INTERFACE I_Cyl_Diag

METHOD M_Diag : E_Diag
VAR_INPUT
END_VAR
END_METHOD

END_INTERFACE

(* stored: Version 1.1.0.1, ProductVersion 3.1.4024.6
   Itf I_Cyl_Diag: Id {535a78e2-f528-00a7-01bb-3c65507c26f9}
   Method M_Diag: Id {2e833c79-50b1-07fc-1bf3-526929dec234} *)
